PROGRAM MAIN
VAR
    initCh1Done : BOOL;
    initCh2Done : BOOL;
    fbNimServo : FB_NimServo;
    fbPd33 : FB_PD33;
    fbVibration : FB_VibrationSensor;

    // DataLogger internal (packed ring buffer)
    logResetLatched : BOOL;
    rec : ARRAY [0..53] OF USINT;
    base : UDINT;
    headMod : UDINT;
    seqLocal : UDINT;
    tUs : UDINT;
    tmpU32 : UDINT;
    tmpI16 : INT;
    tmpI32 : DINT;
    valvesBits : USINT;
END_VAR

GVL_PcDemo.MainCycleCounter := GVL_PcDemo.MainCycleCounter + 1;
GVL_PcDemo.EL3742_Ch2_Sample0_RawCopy := GVL_PcDemo.EL3742_Ch2_Sample0_Raw;

// --- Valve digital outputs (EL2034) ---
IF NOT GVL_ValveIO.Enable THEN
    GVL_ValveIO.Valve1_Cmd := FALSE;
    GVL_ValveIO.Valve2_Cmd := FALSE;
    GVL_ValveIO.Valve3_Cmd := FALSE;
    GVL_ValveIO.Valve4_Cmd := FALSE;
END_IF
GVL_ValveIO.Valve1_Fb := GVL_ValveIO.Valve1_Cmd;
GVL_ValveIO.Valve2_Fb := GVL_ValveIO.Valve2_Cmd;
GVL_ValveIO.Valve3_Fb := GVL_ValveIO.Valve3_Cmd;
GVL_ValveIO.Valve4_Fb := GVL_ValveIO.Valve4_Cmd;

// --- Analog sensors (EL3742) ---
GVL_AnalogSensors.Pressure_RawCopy := GVL_AnalogSensors.Pressure_Raw;
GVL_AnalogSensors.Torque_RawCopy := GVL_AnalogSensors.Torque_Raw;

// Keep EL6022 debug always updated (used by PcHostConsole el6022-dump)
GVL_Rs485Demo.Debug_Ch1_Status := GVL_EL6022_IO.EL6022_Ch1_Status;
GVL_Rs485Demo.Debug_Ch2_Status := GVL_EL6022_IO.EL6022_Ch2_Status;
GVL_Rs485Demo.Debug_Ch1_Ctrl := GVL_EL6022_IO.EL6022_Ch1_Ctrl;
GVL_Rs485Demo.Debug_Ch2_Ctrl := GVL_EL6022_IO.EL6022_Ch2_Ctrl;

// --- NiMotion servo (Modbus RTU over EL6022 / RS-485) ---
fbNimServo(
    Enable := GVL_NimServo.Enable,
    Channel := GVL_NimServo.Channel,
    SlaveId := GVL_NimServo.SlaveId,
    AutoSetCia402Mode := GVL_NimServo.AutoSetCia402Mode,
    DesiredMode := GVL_NimServo.DesiredMode,
    PowerEnable := GVL_NimServo.PowerEnable,
    TargetVelocity := GVL_NimServo.TargetVelocity,
    WordSwap32 := GVL_NimServo.WordSwap32,
    TestForceVelocityWrite := GVL_NimServo.TestForceVelocityWrite,
    ExtendedPoll := GVL_NimServo.ExtendedPoll,
    ApplyVmConfig := GVL_NimServo.ApplyVmConfig,
    VmSpeedMinRpm := GVL_NimServo.VmSpeedMinRpm,
    VmSpeedMaxRpm := GVL_NimServo.VmSpeedMaxRpm,
    VmAccelRpm := GVL_NimServo.VmAccelRpm,
    VmAccelTimeS := GVL_NimServo.VmAccelTimeS,
    VmDecelRpm := GVL_NimServo.VmDecelRpm,
    VmDecelTimeS := GVL_NimServo.VmDecelTimeS,
    CmdSeq := GVL_NimServo.CmdSeq,
    Cmd := GVL_NimServo.Cmd
);

GVL_NimServo.CmdAckSeq := fbNimServo.CmdAckSeq;
GVL_NimServo.Busy := fbNimServo.Busy;
GVL_NimServo.CommOk := fbNimServo.CommOk;
GVL_NimServo.CommErrorCount := fbNimServo.CommErrorCount;
GVL_NimServo.LastErrorId := fbNimServo.LastErrorId;
GVL_NimServo.ControlMode := fbNimServo.ControlMode;
GVL_NimServo.ControlModeOk := fbNimServo.ControlModeOk;
GVL_NimServo.StatusWord := fbNimServo.StatusWord;
GVL_NimServo.ControlWord := fbNimServo.ControlWord;
GVL_NimServo.Cia402State := fbNimServo.Cia402State;
GVL_NimServo.ErrorRegister := fbNimServo.ErrorRegister;
GVL_NimServo.CurrentAlarm := fbNimServo.CurrentAlarm;
GVL_NimServo.DiSignals := fbNimServo.DiSignals;
GVL_NimServo.DoSignals := fbNimServo.DoSignals;
GVL_NimServo.DcBusVoltage := fbNimServo.DcBusVoltage;
GVL_NimServo.ModuleTemp := fbNimServo.ModuleTemp;
GVL_NimServo.Di1Func := fbNimServo.Di1Func;
GVL_NimServo.Di1Logic := fbNimServo.Di1Logic;
GVL_NimServo.Di2Func := fbNimServo.Di2Func;
GVL_NimServo.Di2Logic := fbNimServo.Di2Logic;
GVL_NimServo.Di3Func := fbNimServo.Di3Func;
GVL_NimServo.Di3Logic := fbNimServo.Di3Logic;
GVL_NimServo.Di4Func := fbNimServo.Di4Func;
GVL_NimServo.Di4Logic := fbNimServo.Di4Logic;
GVL_NimServo.Di5Func := fbNimServo.Di5Func;
GVL_NimServo.Di5Logic := fbNimServo.Di5Logic;
GVL_NimServo.Di6Func := fbNimServo.Di6Func;
GVL_NimServo.Di6Logic := fbNimServo.Di6Logic;
GVL_NimServo.Di7Func := fbNimServo.Di7Func;
GVL_NimServo.Di7Logic := fbNimServo.Di7Logic;
GVL_NimServo.Di8Func := fbNimServo.Di8Func;
GVL_NimServo.Di8Logic := fbNimServo.Di8Logic;
GVL_NimServo.Di9Func := fbNimServo.Di9Func;
GVL_NimServo.Di9Logic := fbNimServo.Di9Logic;
GVL_NimServo.EnableDiIndex := fbNimServo.EnableDiIndex;
GVL_NimServo.EnableDiRequired := fbNimServo.EnableDiRequired;
GVL_NimServo.EnableDiActive := fbNimServo.EnableDiActive;
GVL_NimServo.EnableDiOk := fbNimServo.EnableDiOk;
GVL_NimServo.DriveInternalState := fbNimServo.DriveInternalState;
GVL_NimServo.FpgaSystemStatus := fbNimServo.FpgaSystemStatus;
GVL_NimServo.FpgaSystemFault := fbNimServo.FpgaSystemFault;
GVL_NimServo.EncoderInternalFault := fbNimServo.EncoderInternalFault;
GVL_NimServo.FaultRecord := fbNimServo.FaultRecord;
GVL_NimServo.AbsEncoderWord := fbNimServo.AbsEncoderWord;
GVL_NimServo.ModeDisplay := fbNimServo.ModeDisplay;
GVL_NimServo.ActualVelocity := fbNimServo.ActualVelocity;
GVL_NimServo.ActualPosition := fbNimServo.ActualPosition;
GVL_NimServo.CurrentFeedback := fbNimServo.CurrentFeedback;
GVL_NimServo.VmTargetSpeedRpm := fbNimServo.VmTargetSpeedRpm;
GVL_NimServo.VmTargetSpeedEffRpm := fbNimServo.VmTargetSpeedEffRpm;
GVL_NimServo.VmActualSpeedRpm := fbNimServo.VmActualSpeedRpm;
GVL_NimServo.VmCfgPending := fbNimServo.VmCfgPendingOut;
GVL_NimServo.VmCfgIndex := fbNimServo.VmCfgIndexOut;
GVL_NimServo.LastTxLen := fbNimServo.LastTxLen;
GVL_NimServo.LastTx := fbNimServo.LastTx;
GVL_NimServo.LastRxLen := fbNimServo.LastRxLen;
GVL_NimServo.LastRx := fbNimServo.LastRx;

// --- PD33 laser displacement sensor (Modbus RTU over EL6022 / RS-485) ---
GVL_PD33.ChannelConflict := GVL_PD33.Enable AND GVL_NimServo.Enable AND (GVL_PD33.Channel = GVL_NimServo.Channel);
fbPd33(
    Enable := GVL_PD33.Enable AND (NOT GVL_PD33.ChannelConflict),
    Channel := GVL_PD33.Channel,
    SlaveId := GVL_PD33.SlaveId,
    WordSwap32 := GVL_PD33.WordSwap32,
    UseDisplayRegister3B := GVL_PD33.UseDisplayRegister3B,
    CmdSeq := GVL_PD33.CmdSeq,
    Cmd := GVL_PD33.Cmd
);
GVL_PD33.CmdAckSeq := fbPd33.CmdAckSeq;
GVL_PD33.Busy := fbPd33.Busy;
GVL_PD33.PortReady := fbPd33.PortReady;
GVL_PD33.CommOk := fbPd33.CommOk;
GVL_PD33.CommErrorCount := fbPd33.CommErrorCount;
GVL_PD33.LastErrorId := fbPd33.LastErrorId;
GVL_PD33.ExceptionCode := fbPd33.ExceptionCode;
GVL_PD33.RxDiscardCount := fbPd33.RxDiscardCount;
GVL_PD33.LastDiscardId := fbPd33.LastDiscardId;
GVL_PD33.AbsRaw := fbPd33.AbsRaw;
GVL_PD33.RelRaw := fbPd33.RelRaw;
GVL_PD33.AbsMm := fbPd33.AbsMm;
GVL_PD33.RelMm := fbPd33.RelMm;
GVL_PD33.ZeroWord := fbPd33.ZeroWord;
GVL_PD33.LastTxLen := fbPd33.LastTxLen;
GVL_PD33.LastTx := fbPd33.LastTx;
GVL_PD33.LastRxLen := fbPd33.LastRxLen;
GVL_PD33.LastRx := fbPd33.LastRx;

// --- VB02 vibration sensor (Modbus RTU over EL6022 Ch2 / RS-485) ---
fbVibration(
    Enable := GVL_Vibration.Enable,
    Channel := GVL_Vibration.Channel,
    SlaveId := GVL_Vibration.SlaveId,
    MinGapMs := GVL_Vibration.MinGapMs,
    TimeoutMs := GVL_Vibration.TimeoutMs
);
GVL_Vibration.Busy := fbVibration.Busy;
GVL_Vibration.PortReady := fbVibration.PortReady;
GVL_Vibration.CommOk := fbVibration.CommOk;
GVL_Vibration.CommErrorCount := fbVibration.CommErrorCount;
GVL_Vibration.LastErrorId := fbVibration.LastErrorId;
GVL_Vibration.ExceptionCode := fbVibration.ExceptionCode;
GVL_Vibration.RxDiscardCount := fbVibration.RxDiscardCount;
GVL_Vibration.LastDiscardId := fbVibration.LastDiscardId;
GVL_Vibration.SampleSeq := fbVibration.SampleSeq;
GVL_Vibration.AccXRaw := fbVibration.AccXRaw;
GVL_Vibration.AccYRaw := fbVibration.AccYRaw;
GVL_Vibration.AccZRaw := fbVibration.AccZRaw;
GVL_Vibration.VelXRaw := fbVibration.VelXRaw;
GVL_Vibration.VelYRaw := fbVibration.VelYRaw;
GVL_Vibration.VelZRaw := fbVibration.VelZRaw;
GVL_Vibration.TempRaw := fbVibration.TempRaw;
GVL_Vibration.DispXRaw := fbVibration.DispXRaw;
GVL_Vibration.DispYRaw := fbVibration.DispYRaw;
GVL_Vibration.DispZRaw := fbVibration.DispZRaw;
GVL_Vibration.FreqXRaw := fbVibration.FreqXRaw;
GVL_Vibration.FreqYRaw := fbVibration.FreqYRaw;
GVL_Vibration.FreqZRaw := fbVibration.FreqZRaw;
GVL_Vibration.AccX := fbVibration.AccX;
GVL_Vibration.AccY := fbVibration.AccY;
GVL_Vibration.AccZ := fbVibration.AccZ;
GVL_Vibration.VelX := fbVibration.VelX;
GVL_Vibration.VelY := fbVibration.VelY;
GVL_Vibration.VelZ := fbVibration.VelZ;
GVL_Vibration.TempC := fbVibration.TempC;
GVL_Vibration.DispX := fbVibration.DispX;
GVL_Vibration.DispY := fbVibration.DispY;
GVL_Vibration.DispZ := fbVibration.DispZ;
GVL_Vibration.FreqX := fbVibration.FreqX;
GVL_Vibration.FreqY := fbVibration.FreqY;
GVL_Vibration.FreqZ := fbVibration.FreqZ;
GVL_Vibration.LastTxLen := fbVibration.LastTxLen;
GVL_Vibration.LastTx := fbVibration.LastTx;
GVL_Vibration.LastRxLen := fbVibration.LastRxLen;
GVL_Vibration.LastRx := fbVibration.LastRx;
// --- DataLogger ring buffer (packed bytes) ---
// Time base: PlcTask cycle is 2000us (see PlcTask.TcTTO). Use cycle counter for monotonic time.
tUs := ULINT_TO_UDINT(GVL_PcDemo.MainCycleCounter) * 2000;

IF GVL_DataLogger.Reset AND (NOT logResetLatched) THEN
    logResetLatched := TRUE;
    GVL_DataLogger.Head := 0;
    GVL_DataLogger.Tail := 0;
    GVL_DataLogger.Seq := 0;
    GVL_DataLogger.OverrunCount := 0;
    GVL_DataLogger.DropCount := 0;
ELSIF (NOT GVL_DataLogger.Reset) THEN
    logResetLatched := FALSE;
END_IF

IF GVL_DataLogger.Enable THEN
    // Overrun detection: if head - tail > BufferSize - RecordSize, drop this sample.
    IF (GVL_DataLogger.Head - GVL_DataLogger.Tail) > (GVL_DataLogger.BufferSize - GVL_DataLogger.RecordSize) THEN
        GVL_DataLogger.OverrunCount := GVL_DataLogger.OverrunCount + 1;
    ELSE
        seqLocal := GVL_DataLogger.Seq;

        // magic 'VBM1' = 0x56424D31
        rec[0] := 16#31; rec[1] := 16#4D; rec[2] := 16#42; rec[3] := 16#56;

        // seq (u32)
        tmpU32 := seqLocal;
        rec[4] := UDINT_TO_USINT(tmpU32 AND 16#FF);
        rec[5] := UDINT_TO_USINT(SHR(tmpU32, 8) AND 16#FF);
        rec[6] := UDINT_TO_USINT(SHR(tmpU32, 16) AND 16#FF);
        rec[7] := UDINT_TO_USINT(SHR(tmpU32, 24) AND 16#FF);

        // t_us (u32)
        tmpU32 := tUs;
        rec[8] := UDINT_TO_USINT(tmpU32 AND 16#FF);
        rec[9] := UDINT_TO_USINT(SHR(tmpU32, 8) AND 16#FF);
        rec[10] := UDINT_TO_USINT(SHR(tmpU32, 16) AND 16#FF);
        rec[11] := UDINT_TO_USINT(SHR(tmpU32, 24) AND 16#FF);

        // pressure_raw (i16)
        tmpI16 := GVL_AnalogSensors.Pressure_RawCopy;
        tmpU32 := INT_TO_UDINT(tmpI16) AND 16#FFFF;
        rec[12] := UDINT_TO_USINT(tmpU32 AND 16#FF);
        rec[13] := UDINT_TO_USINT(SHR(tmpU32, 8) AND 16#FF);

        // torque_raw (i16)
        tmpI16 := GVL_AnalogSensors.Torque_RawCopy;
        tmpU32 := INT_TO_UDINT(tmpI16) AND 16#FFFF;
        rec[14] := UDINT_TO_USINT(tmpU32 AND 16#FF);
        rec[15] := UDINT_TO_USINT(SHR(tmpU32, 8) AND 16#FF);

        // pd33_abs_raw (i32)
        tmpI32 := GVL_PD33.AbsRaw;
        tmpU32 := DINT_TO_UDINT(tmpI32);
        rec[16] := UDINT_TO_USINT(tmpU32 AND 16#FF);
        rec[17] := UDINT_TO_USINT(SHR(tmpU32, 8) AND 16#FF);
        rec[18] := UDINT_TO_USINT(SHR(tmpU32, 16) AND 16#FF);
        rec[19] := UDINT_TO_USINT(SHR(tmpU32, 24) AND 16#FF);

        // pd33_rel_raw (i32)
        tmpI32 := GVL_PD33.RelRaw;
        tmpU32 := DINT_TO_UDINT(tmpI32);
        rec[20] := UDINT_TO_USINT(tmpU32 AND 16#FF);
        rec[21] := UDINT_TO_USINT(SHR(tmpU32, 8) AND 16#FF);
        rec[22] := UDINT_TO_USINT(SHR(tmpU32, 16) AND 16#FF);
        rec[23] := UDINT_TO_USINT(SHR(tmpU32, 24) AND 16#FF);

        // vibration raw values (i16)
        tmpI16 := GVL_Vibration.AccXRaw;
        tmpU32 := INT_TO_UDINT(tmpI16) AND 16#FFFF;
        rec[24] := UDINT_TO_USINT(tmpU32 AND 16#FF);
        rec[25] := UDINT_TO_USINT(SHR(tmpU32, 8) AND 16#FF);

        tmpI16 := GVL_Vibration.AccYRaw;
        tmpU32 := INT_TO_UDINT(tmpI16) AND 16#FFFF;
        rec[26] := UDINT_TO_USINT(tmpU32 AND 16#FF);
        rec[27] := UDINT_TO_USINT(SHR(tmpU32, 8) AND 16#FF);

        tmpI16 := GVL_Vibration.AccZRaw;
        tmpU32 := INT_TO_UDINT(tmpI16) AND 16#FFFF;
        rec[28] := UDINT_TO_USINT(tmpU32 AND 16#FF);
        rec[29] := UDINT_TO_USINT(SHR(tmpU32, 8) AND 16#FF);

        tmpI16 := GVL_Vibration.VelXRaw;
        tmpU32 := INT_TO_UDINT(tmpI16) AND 16#FFFF;
        rec[30] := UDINT_TO_USINT(tmpU32 AND 16#FF);
        rec[31] := UDINT_TO_USINT(SHR(tmpU32, 8) AND 16#FF);

        tmpI16 := GVL_Vibration.VelYRaw;
        tmpU32 := INT_TO_UDINT(tmpI16) AND 16#FFFF;
        rec[32] := UDINT_TO_USINT(tmpU32 AND 16#FF);
        rec[33] := UDINT_TO_USINT(SHR(tmpU32, 8) AND 16#FF);

        tmpI16 := GVL_Vibration.VelZRaw;
        tmpU32 := INT_TO_UDINT(tmpI16) AND 16#FFFF;
        rec[34] := UDINT_TO_USINT(tmpU32 AND 16#FF);
        rec[35] := UDINT_TO_USINT(SHR(tmpU32, 8) AND 16#FF);

        tmpI16 := GVL_Vibration.TempRaw;
        tmpU32 := INT_TO_UDINT(tmpI16) AND 16#FFFF;
        rec[36] := UDINT_TO_USINT(tmpU32 AND 16#FF);
        rec[37] := UDINT_TO_USINT(SHR(tmpU32, 8) AND 16#FF);

        tmpI16 := GVL_Vibration.DispXRaw;
        tmpU32 := INT_TO_UDINT(tmpI16) AND 16#FFFF;
        rec[38] := UDINT_TO_USINT(tmpU32 AND 16#FF);
        rec[39] := UDINT_TO_USINT(SHR(tmpU32, 8) AND 16#FF);

        tmpI16 := GVL_Vibration.DispYRaw;
        tmpU32 := INT_TO_UDINT(tmpI16) AND 16#FFFF;
        rec[40] := UDINT_TO_USINT(tmpU32 AND 16#FF);
        rec[41] := UDINT_TO_USINT(SHR(tmpU32, 8) AND 16#FF);

        tmpI16 := GVL_Vibration.DispZRaw;
        tmpU32 := INT_TO_UDINT(tmpI16) AND 16#FFFF;
        rec[42] := UDINT_TO_USINT(tmpU32 AND 16#FF);
        rec[43] := UDINT_TO_USINT(SHR(tmpU32, 8) AND 16#FF);

        tmpI16 := GVL_Vibration.FreqXRaw;
        tmpU32 := INT_TO_UDINT(tmpI16) AND 16#FFFF;
        rec[44] := UDINT_TO_USINT(tmpU32 AND 16#FF);
        rec[45] := UDINT_TO_USINT(SHR(tmpU32, 8) AND 16#FF);

        tmpI16 := GVL_Vibration.FreqYRaw;
        tmpU32 := INT_TO_UDINT(tmpI16) AND 16#FFFF;
        rec[46] := UDINT_TO_USINT(tmpU32 AND 16#FF);
        rec[47] := UDINT_TO_USINT(SHR(tmpU32, 8) AND 16#FF);

        tmpI16 := GVL_Vibration.FreqZRaw;
        tmpU32 := INT_TO_UDINT(tmpI16) AND 16#FFFF;
        rec[48] := UDINT_TO_USINT(tmpU32 AND 16#FF);
        rec[49] := UDINT_TO_USINT(SHR(tmpU32, 8) AND 16#FF);
        // valves bits
        valvesBits := 0;
        IF GVL_ValveIO.Valve1_Fb THEN valvesBits := valvesBits OR 16#01; END_IF
        IF GVL_ValveIO.Valve2_Fb THEN valvesBits := valvesBits OR 16#02; END_IF
        IF GVL_ValveIO.Valve3_Fb THEN valvesBits := valvesBits OR 16#04; END_IF
        IF GVL_ValveIO.Valve4_Fb THEN valvesBits := valvesBits OR 16#08; END_IF
        rec[50] := valvesBits;

        // flags
        rec[51] := 0;
        IF GVL_PD33.CommOk THEN rec[51] := rec[51] OR 16#01; END_IF
        IF GVL_Vibration.CommOk THEN rec[51] := rec[51] OR 16#02; END_IF

        // reserved u16
        rec[52] := 0;
        rec[53] := 0;

        // write record into ring (buffer size is multiple of record size)
        headMod := GVL_DataLogger.Head MOD GVL_DataLogger.BufferSize;
        base := headMod;
        GVL_DataLogger.Buffer[base + 0] := rec[0];
        GVL_DataLogger.Buffer[base + 1] := rec[1];
        GVL_DataLogger.Buffer[base + 2] := rec[2];
        GVL_DataLogger.Buffer[base + 3] := rec[3];
        GVL_DataLogger.Buffer[base + 4] := rec[4];
        GVL_DataLogger.Buffer[base + 5] := rec[5];
        GVL_DataLogger.Buffer[base + 6] := rec[6];
        GVL_DataLogger.Buffer[base + 7] := rec[7];
        GVL_DataLogger.Buffer[base + 8] := rec[8];
        GVL_DataLogger.Buffer[base + 9] := rec[9];
        GVL_DataLogger.Buffer[base + 10] := rec[10];
        GVL_DataLogger.Buffer[base + 11] := rec[11];
        GVL_DataLogger.Buffer[base + 12] := rec[12];
        GVL_DataLogger.Buffer[base + 13] := rec[13];
        GVL_DataLogger.Buffer[base + 14] := rec[14];
        GVL_DataLogger.Buffer[base + 15] := rec[15];
        GVL_DataLogger.Buffer[base + 16] := rec[16];
        GVL_DataLogger.Buffer[base + 17] := rec[17];
        GVL_DataLogger.Buffer[base + 18] := rec[18];
        GVL_DataLogger.Buffer[base + 19] := rec[19];
        GVL_DataLogger.Buffer[base + 20] := rec[20];
        GVL_DataLogger.Buffer[base + 21] := rec[21];
        GVL_DataLogger.Buffer[base + 22] := rec[22];
        GVL_DataLogger.Buffer[base + 23] := rec[23];
        GVL_DataLogger.Buffer[base + 24] := rec[24];
        GVL_DataLogger.Buffer[base + 25] := rec[25];
        GVL_DataLogger.Buffer[base + 26] := rec[26];
        GVL_DataLogger.Buffer[base + 27] := rec[27];
        GVL_DataLogger.Buffer[base + 28] := rec[28];
        GVL_DataLogger.Buffer[base + 29] := rec[29];
        GVL_DataLogger.Buffer[base + 30] := rec[30];
        GVL_DataLogger.Buffer[base + 31] := rec[31];
        GVL_DataLogger.Buffer[base + 32] := rec[32];
        GVL_DataLogger.Buffer[base + 33] := rec[33];
        GVL_DataLogger.Buffer[base + 34] := rec[34];
        GVL_DataLogger.Buffer[base + 35] := rec[35];
        GVL_DataLogger.Buffer[base + 36] := rec[36];
        GVL_DataLogger.Buffer[base + 37] := rec[37];
        GVL_DataLogger.Buffer[base + 38] := rec[38];
        GVL_DataLogger.Buffer[base + 39] := rec[39];
        GVL_DataLogger.Buffer[base + 40] := rec[40];
        GVL_DataLogger.Buffer[base + 41] := rec[41];
        GVL_DataLogger.Buffer[base + 42] := rec[42];
        GVL_DataLogger.Buffer[base + 43] := rec[43];
        GVL_DataLogger.Buffer[base + 44] := rec[44];
        GVL_DataLogger.Buffer[base + 45] := rec[45];
        GVL_DataLogger.Buffer[base + 46] := rec[46];
        GVL_DataLogger.Buffer[base + 47] := rec[47];
        GVL_DataLogger.Buffer[base + 48] := rec[48];
        GVL_DataLogger.Buffer[base + 49] := rec[49];
        GVL_DataLogger.Buffer[base + 50] := rec[50];
        GVL_DataLogger.Buffer[base + 51] := rec[51];
        GVL_DataLogger.Buffer[base + 52] := rec[52];
        GVL_DataLogger.Buffer[base + 53] := rec[53];

        GVL_DataLogger.Head := GVL_DataLogger.Head + GVL_DataLogger.RecordSize;
        GVL_DataLogger.Seq := GVL_DataLogger.Seq + 1;
    END_IF
END_IF

IF (NOT GVL_NimServo.Enable) AND (NOT GVL_PD33.Enable) AND (NOT GVL_Vibration.Enable) AND GVL_Rs485Demo.Enable THEN
// --- EL6022 RS-485 demo loopback (Ch1 <-> Ch2) ---
// One-time init handshake (Ctrl bit2 / Status bit2)
IF NOT initCh1Done THEN
    GVL_EL6022_IO.EL6022_Ch1_Ctrl := GVL_EL6022_IO.EL6022_Ch1_Ctrl OR 16#0004;
    IF (GVL_EL6022_IO.EL6022_Ch1_Status AND 16#0004) <> 0 THEN
        GVL_EL6022_IO.EL6022_Ch1_Ctrl := GVL_EL6022_IO.EL6022_Ch1_Ctrl AND 16#FFFB;
        initCh1Done := TRUE;
    END_IF
END_IF

IF NOT initCh2Done THEN
    GVL_EL6022_IO.EL6022_Ch2_Ctrl := GVL_EL6022_IO.EL6022_Ch2_Ctrl OR 16#0004;
    IF (GVL_EL6022_IO.EL6022_Ch2_Status AND 16#0004) <> 0 THEN
        GVL_EL6022_IO.EL6022_Ch2_Ctrl := GVL_EL6022_IO.EL6022_Ch2_Ctrl AND 16#FFFB;
        initCh2Done := TRUE;
    END_IF
END_IF

// TX handshake: low byte bits: b0=TxReq, b1=RxAck, b2=InitReq, b3=SendContinuous, high byte = length
IF (GVL_Rs485Demo.TxBusy = FALSE) AND (GVL_Rs485Demo.TxSeq <> GVL_Rs485Demo.TxDoneSeq) THEN
    // Prepare control word for selected TX channel
    IF GVL_Rs485Demo.TxUseCh2 THEN
        // Copy TX payload
        GVL_EL6022_IO.EL6022_Ch2_DataOut := GVL_Rs485Demo.TxData;
        // Set length (high byte) and TxReq (bit0)
        GVL_EL6022_IO.EL6022_Ch2_Ctrl := (GVL_EL6022_IO.EL6022_Ch2_Ctrl AND 16#00FF) OR 16#0001 OR SHL(USINT_TO_WORD(GVL_Rs485Demo.TxLen), 8);
    ELSE
        GVL_EL6022_IO.EL6022_Ch1_DataOut := GVL_Rs485Demo.TxData;
        GVL_EL6022_IO.EL6022_Ch1_Ctrl := (GVL_EL6022_IO.EL6022_Ch1_Ctrl AND 16#00FF) OR 16#0001 OR SHL(USINT_TO_WORD(GVL_Rs485Demo.TxLen), 8);
    END_IF

    GVL_Rs485Demo.TxBusy := TRUE;
END_IF

// Observe Tx accepted on the selected channel (Status bit0)
IF GVL_Rs485Demo.TxBusy THEN
    IF GVL_Rs485Demo.TxUseCh2 THEN
        IF (GVL_EL6022_IO.EL6022_Ch2_Status AND 16#0001) <> 0 THEN
            // Clear TxReq bit after accepted
            GVL_EL6022_IO.EL6022_Ch2_Ctrl := GVL_EL6022_IO.EL6022_Ch2_Ctrl AND 16#00FE;
            GVL_Rs485Demo.TxDoneSeq := GVL_Rs485Demo.TxSeq;
            GVL_Rs485Demo.TxBusy := FALSE;
        END_IF
    ELSE
        IF (GVL_EL6022_IO.EL6022_Ch1_Status AND 16#0001) <> 0 THEN
            GVL_EL6022_IO.EL6022_Ch1_Ctrl := GVL_EL6022_IO.EL6022_Ch1_Ctrl AND 16#00FE;
            GVL_Rs485Demo.TxDoneSeq := GVL_Rs485Demo.TxSeq;
            GVL_Rs485Demo.TxBusy := FALSE;
        END_IF
    END_IF
END_IF

// RX handling: Status bit1=Receive request, high byte = input length
IF (GVL_EL6022_IO.EL6022_Ch1_Status AND 16#0002) <> 0 THEN
    GVL_Rs485Demo.RxFromCh2 := FALSE;
    GVL_Rs485Demo.RxStatus := GVL_EL6022_IO.EL6022_Ch1_Status;
    GVL_Rs485Demo.RxLen := WORD_TO_USINT(SHR(GVL_EL6022_IO.EL6022_Ch1_Status, 8));
    GVL_Rs485Demo.RxData := GVL_EL6022_IO.EL6022_Ch1_DataIn;
    GVL_Rs485Demo.RxSeq := GVL_Rs485Demo.RxSeq + 1;
    // Acknowledge receive (Ctrl bit1)
    GVL_EL6022_IO.EL6022_Ch1_Ctrl := GVL_EL6022_IO.EL6022_Ch1_Ctrl OR 16#0002;
ELSIF (GVL_EL6022_IO.EL6022_Ch2_Status AND 16#0002) <> 0 THEN
    GVL_Rs485Demo.RxFromCh2 := TRUE;
    GVL_Rs485Demo.RxStatus := GVL_EL6022_IO.EL6022_Ch2_Status;
    GVL_Rs485Demo.RxLen := WORD_TO_USINT(SHR(GVL_EL6022_IO.EL6022_Ch2_Status, 8));
    GVL_Rs485Demo.RxData := GVL_EL6022_IO.EL6022_Ch2_DataIn;
    GVL_Rs485Demo.RxSeq := GVL_Rs485Demo.RxSeq + 1;
    GVL_EL6022_IO.EL6022_Ch2_Ctrl := GVL_EL6022_IO.EL6022_Ch2_Ctrl OR 16#0002;
ELSE
    // Drop RxAck bits when no receive request pending
    GVL_EL6022_IO.EL6022_Ch1_Ctrl := GVL_EL6022_IO.EL6022_Ch1_Ctrl AND 16#FFFD;
    GVL_EL6022_IO.EL6022_Ch2_Ctrl := GVL_EL6022_IO.EL6022_Ch2_Ctrl AND 16#FFFD;
END_IF
END_IF

END_PROGRAM

(* stored: Version 1.1.0.1, ProductVersion 3.1.4024.13
   POU MAIN: Id {7d47c4d8-afbc-4278-8b7f-8e4ca1a04aee}, SpecialFunc None *)
